// TIA Portal V16 export
// export: Created 2025-12-30T17:36:41.5072322Z, ExportSetting WithDefaults, DisplayName Totally Integrated Automation Portal, DisplayVersion V16, DisplayName TIA Portal Version Control Interface, DisplayVersion V16, DisplayName TIA Portal Openness, DisplayVersion V16, DisplayName STEP 7 Professional, DisplayVersion V16, DisplayName STEP 7 Safety, DisplayVersion V16, DisplayName WinCC Professional, DisplayVersion V16
VAR_GLOBAL   // PLC tag table "Standard-Variablentabelle"
   Clock_Byte AT %MB1 : Byte;
   Clock_10Hz AT %M1.0 : Bool;
   Clock_5Hz AT %M1.1 : Bool;
   "Clock_2.5Hz" AT %M1.2 : Bool;
   Clock_2Hz AT %M1.3 : Bool;
   "Clock_1.25Hz" AT %M1.4 : Bool;
   Clock_1Hz AT %M1.5 : Bool;
   "Clock_0.625Hz" AT %M1.6 : Bool;
   "Clock_0.5Hz" AT %M1.7 : Bool;
   "Reset Coutner" AT %I2.0 : Bool;
   "Reset Coutner Light" AT %Q1.4 : Bool;
END_VAR
